FUNCTION_BLOCK FB_HeatingNetworkLowTemperature
VAR_INPUT
	ambientState : ST_AmbientState;
	
	//control struct for hnlt
	controlAutomatic : ST_HeatingNetworkLowTemperatureControl;	
END_VAR
VAR_OUTPUT
	{attribute 'OPC.UA.DA' := '1'}
	localState : ST_BufferStorageState;
END_VAR
VAR
	//systems
	BufferStorage : FB_BufferStorage;
	OuterCapillaryTubeMats : FB_OuterCapillaryTubeMats;
	HVFASystem : FB_HVFAStorageSystem;
	CompressorSystem : FB_CompressorSystem;
	AnnealingOvenSealingSystem : FB_AnnealingOvenSealingSystem;
	DCSystem : FB_DCSystem;
	
	//machines
	AnnealingOvenSealing : FB_AnnealingOven;
	DC : FB_DC;

	//internal variables
	fSetPoint_HVFASystem : REAL;
	bSetStatusOn_AnnealingOven : BOOL;
	bSetStatusOn_DC : BOOL;
END_VAR

//buffer storage system
BufferStorage();
localState := BufferStorage.localState;

//producer
CompressorSystem(bSetStatusOnAutomatic := TRUE,
	bAlgorithmPermission := controlAutomatic.bAlgorithmPermission,
	fSetPointAutomatic := controlAutomatic.fFeedTemperature_Heating);

//consumer
OuterCapillaryTubeMats(bSetStatusOnAutomatic := controlAutomatic.bSetStatusOn_OuterCapillaryTubeMats,
	bAlgorithmPermission := controlAutomatic.bAlgorithmPermission,
	fSetPointAutomatic := controlAutomatic.fFeedTemperature_Cooling,
	stAmbientState := ambientState);
	
AnnealingOvenSealing();
bSetStatusOn_AnnealingOven := AnnealingOvenSealing.bStatusOn_Sealing;
AnnealingOvenSealingSystem(bSetStatusOnAutomatic := bSetStatusOn_AnnealingOven,
	bAlgorithmPermission := controlAutomatic.bAlgorithmPermission,
	fSetPointAutomatic := 35);
	
DC();
bSetStatusOn_DC := DC.bStatusOn;
DCSystem(bSetStatusOnAutomatic := bSetStatusOn_DC,
	bAlgorithmPermission := controlAutomatic.bAlgorithmPermission,
	fSetPointAutomatic := 35);

//external storages
//setpoint depends on loading mode -> storage must be warmer than setpoint temperature in network
IF controlAutomatic.bLoading_HVFASystem THEN
	fSetPoint_HVFASystem := controlAutomatic.fFeedTemperature_Heating+5;
ELSE
	fSetPoint_HVFASystem := controlAutomatic.fFeedTemperature_Heating;
END_IF
HVFASystem(bSetStatusOnAutomatic := controlAutomatic.bSetStatusOn_HVFASystem,
	bAlgorithmPermission := controlAutomatic.bAlgorithmPermission,
	fSetPointAutomatic := fSetpoint_HVFASystem,
	bLoadingAutomatic := controlAutomatic.bLoading_HVFASystem,
	aTelegramm_WMZ7x0 := aTelegramm_WMZ720,
	aTelegramm_WMZx05 := aTelegramm_WMZ205);

END_FUNCTION_BLOCK

(* stored: Version 1.1.0.1, ProductVersion 3.1.4024.10
   POU FB_HeatingNetworkLowTemperature: Id {41e3edb3-66e7-411c-a35e-b44e9a5d66f1}, SpecialFunc None *)
